// TIA Portal V16 export
// export: Created 2022-11-17T15:49:50.2761183Z, ExportSetting WithDefaults, DisplayName Totally Integrated Automation Portal, DisplayVersion V16 Update 6, DisplayName TIA Portal Version Control Interface, DisplayVersion V16 Update 2, DisplayName TIA Portal Openness, DisplayVersion V16 Update 6, DisplayName SINAMICS Startdrive Advanced, DisplayVersion V16 Update 5, DisplayName SINAMICS Startdrive G130, G150, S120, S150, SINAMICS MV, S210, DisplayVersion V16 Update 5, DisplayName SINAMICS Startdrive G110M, G120, G120C, G120D, G120P, G115D, DisplayVersion V16 Update 5, DisplayName STEP 7 Professional, DisplayVersion V16 Update 6, DisplayName STEP 7 Safety, DisplayVersion V16, DisplayName WinCC Advanced, DisplayVersion V16 Update 6
TYPE "InverterData"
// stored: IsFailsafeCompliant false
   STRUCT
      control_word : Word;
      setpoint : Real;
      ref_quantity : Struct
         speed_p2000 : Real;
         current_p2002 : Real;
         torque_p2003 : Real;
      END_STRUCT;
      status_word : Word;
      actual_speed : Real;
      actual_current : Real;
      actual_torque : Real;
      actual_alarm : Word;
      actual_fault : Word;
      RETVAL_RD : Word;
      RETVAL_WR : Word;
   END_STRUCT;
END_TYPE
